(* PLC project Unnamed, Unknown Unnamed 1 *)
(* stored: creationDateTime 2025-11-19T16:38:19, modificationDateTime 2025-11-19T18:11:03 *)

PROGRAM program0
  VAR
    LED AT %QX0.0 : BOOL;
    UP_start AT %IX0.0 : BOOL;
    DOWN_stop AT %IX0.1 : BOOL;
  END_VAR
  VAR
    Latch : BOOL;
  END_VAR

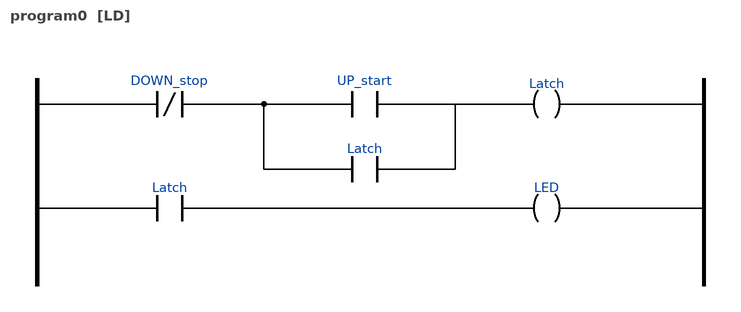
(* LD diagram, written out as Structured Text *)
Latch := NOT DOWN_stop AND (Latch OR UP_start);
LED := Latch;
END_PROGRAM

CONFIGURATION Config0
  VAR_GLOBAL
    LocalVar0 : BOOL;
  END_VAR
  RESOURCE Res0 ON PLC
    TASK task0(INTERVAL := T#20ms, PRIORITY := 0);
    PROGRAM instance0 WITH task0 : program0;
  END_RESOURCE
END_CONFIGURATION
